FUNCTION_BLOCK DrillStation_HCECC (* Model a conveyor *)
  (* Standard: 61499-2 *)
  (* Version 0.2, 2003-12-04, JHC, Rockwell Automation, Renamed for better indexing. *)
  (* Compiler header: package fb.rt.benchmarks.DrillStation; *)
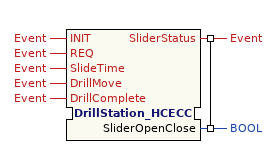
  EVENT_INPUT
    INIT; (* Initialization Request *)
    REQ; (* Normal Execution Request *)
    SlideTime;
    DrillMove;
    DrillComplete;
  END_EVENT
  EVENT_OUTPUT
    SliderStatus WITH SliderOpenClose;
  END_EVENT
  VAR_OUTPUT
    SliderOpenClose : BOOL;
  END_VAR
  VAR
    ReadyNot : BOOL; (* ready: true, not ready: false *)
    OpenClose : BOOL := true; (* true: open, false: close *)
    UP_DOWN : BOOL := true; (* true: up, false: down *)
    DrillStart : BOOL := false;
    DrillDone : BOOL := false;
  END_VAR
  ALGORITHM INITDrill IN ST: (* Initialization algorithm *)
UP_DOWN := TRUE;
  END_ALGORITHM
  ALGORITHM MovingDown IN ST: (* Normally executed algorithm *)
UP_DOWN := FALSE;
DrillStart := FALSE;
  END_ALGORITHM
  ALGORITHM SetDrillDone IN ST: (* Initialization algorithm *)
DrillDone := TRUE;
  END_ALGORITHM
  ALGORITHM INITSlider IN ST: (* Initialization algorithm *)
OpenClose := TRUE;
  END_ALGORITHM
  ALGORITHM REQSlider IN ST: (* Normally executed algorithm *)
OpenClose := FALSE;
  END_ALGORITHM
  ALGORITHM DrillStart IN ST: (* Initialization algorithm *)
DrillStart := TRUE;
  END_ALGORITHM
END_FUNCTION_BLOCK
(* other elements stored in the file *)
(* ECC Name=Drill *)
(* ECState Name=START Comment=Initial State *)
(* ECAction Algorithm=INITDrill *)
(* ECState Name=REQ Comment=Normal execution *)
(* ECAction Algorithm=MovingDown *)
(* ECState Name=Done *)
(* ECAction Algorithm=SetDrillDone *)
(* ECState Name=Drilling *)
(* ECTransition Destination=REQ Source=START Condition=DrillStart *)
(* ECTransition Destination=START Source=Done Condition=DrillMove *)
(* ECTransition Destination=Drilling Source=REQ Condition=DrillMove *)
(* ECTransition Destination=Done Source=Drilling Condition=DrillComplete *)
(* ECC Name=Slider *)
(* ECState Name=START Comment=Initial State *)
(* ECAction Output=SliderStatus Algorithm=INITSlider *)
(* ECState Name=REQ Comment=Normal execution *)
(* ECAction Output=SliderStatus Algorithm=REQSlider *)
(* ECState Name=Drilling *)
(* ECAction Algorithm=DrillStart *)
(* ECState Name=ReturnSlide *)
(* ECState Name=WaitForDrill *)
(* ECTransition Destination=REQ Source=START Condition=REQ *)
(* ECTransition Destination=Drilling Source=REQ Condition=SlideTime *)
(* ECTransition Destination=ReturnSlide Source=Drilling Condition=DrillComplete *)
(* ECTransition Destination=WaitForDrill Source=ReturnSlide Condition=SlideTime *)
(* ECTransition Destination=START Source=WaitForDrill Condition=UP_DOWN *)
